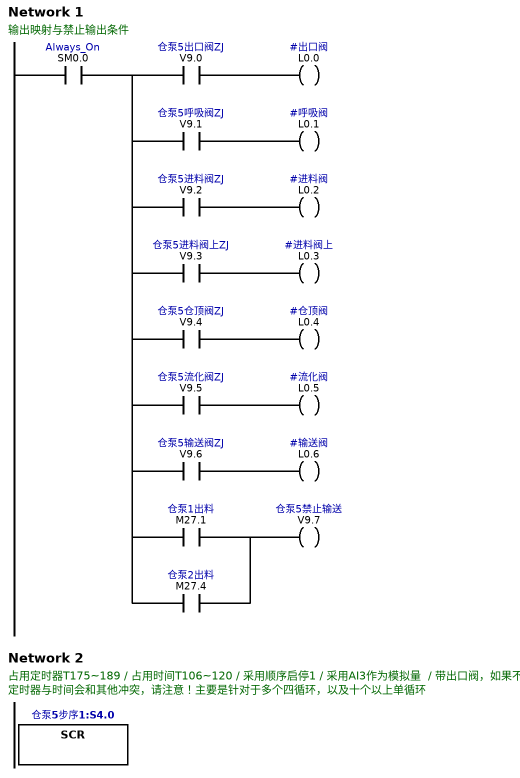
[picture p72: SBR24 networks 1-2]
Network 1
// 输出映射与禁止输出条件
LD     Always_On:SM0.0
LPS
A      仓泵5出口阀ZJ:V9.0
=      #出口阀:L0.0
LRD
A      仓泵5呼吸阀ZJ:V9.1
=      #呼吸阀:L0.1
LRD
A      仓泵5进料阀ZJ:V9.2
=      #进料阀:L0.2
LRD
A      仓泵5进料阀上ZJ:V9.3
=      #进料阀上:L0.3
LRD
A      仓泵5仓顶阀ZJ:V9.4
=      #仓顶阀:L0.4
LRD
A      仓泵5流化阀ZJ:V9.5
=      #流化阀:L0.5
LRD
A      仓泵5输送阀ZJ:V9.6
=      #输送阀:L0.6
LPP
LD     仓泵1出料:M27.1
O      仓泵2出料:M27.4
ALD
=      仓泵5禁止输送:V9.7
Network 2
// 占用定时器T175~189
// 占用时间T106~120
// 采用顺序启停1
// 采用AI3作为模拟量 
// 带出口阀，如果不需要可删除
// 同时仅一个仓泵出料，多需求请改网络5
// 定时器与时间会和其他冲突，请注意！主要是针对于多个四循环，以及十个以上单循环
LSCR   仓泵5步序1:S4.0
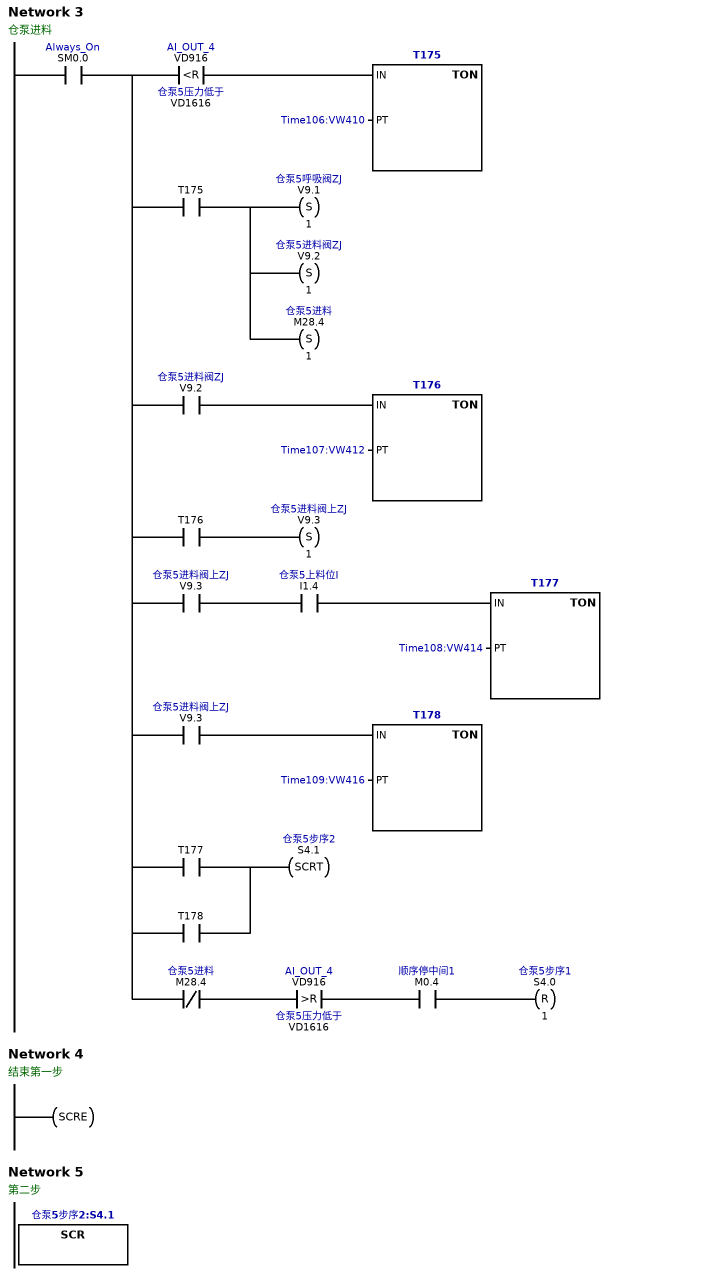
Network 3
// 仓泵进料
LD     Always_On:SM0.0
LPS
AR<    AI_OUT_4:VD916, 仓泵5压力低于:VD1616
TON    T175, Time106:VW410
LRD
A      T175
S      仓泵5呼吸阀ZJ:V9.1, 1
S      仓泵5进料阀ZJ:V9.2, 1
S      仓泵5进料:M28.4, 1
LRD
LPS
A      仓泵5进料阀ZJ:V9.2
TON    T176, Time107:VW412
LRD
A      T176
S      仓泵5进料阀上ZJ:V9.3, 1
LRD
A      仓泵5进料阀上ZJ:V9.3
A      仓泵5上料位I:I1.4
TON    T177, Time108:VW414
LPP
A      仓泵5进料阀上ZJ:V9.3
TON    T178, Time109:VW416
LRD
LD     T177
O      T178
ALD
SCRT   仓泵5步序2:S4.1
LPP
AN     仓泵5进料:M28.4
AR>    AI_OUT_4:VD916, 仓泵5压力低于:VD1616
A      顺序停中间1:M0.4
R      仓泵5步序1:S4.0, 1
Network 4
// 结束第一步
SCRE
Network 5
// 第二步 
LSCR   仓泵5步序2:S4.1
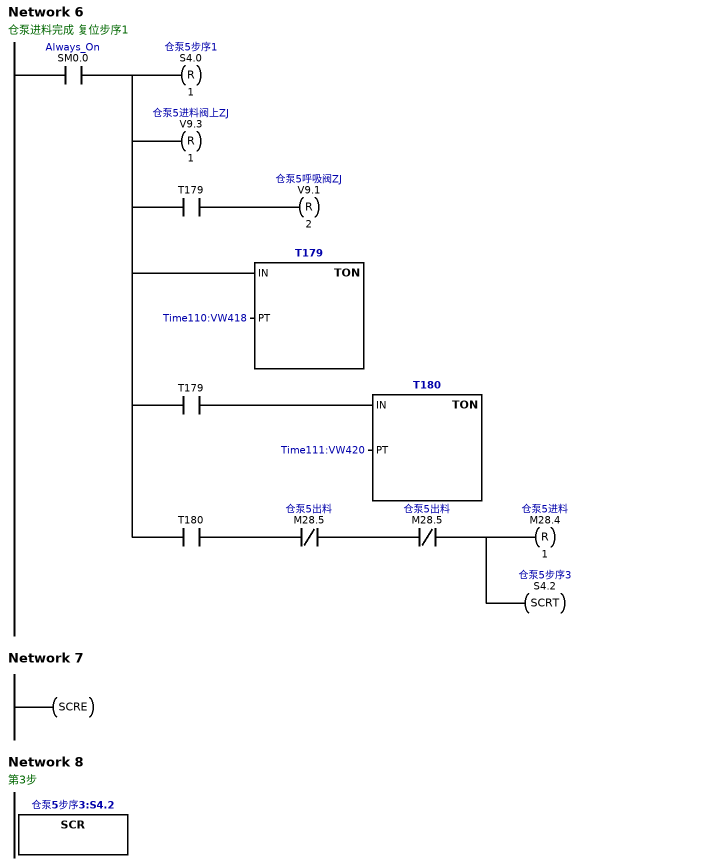
Network 6
// 仓泵进料完成 复位步序1
LD     Always_On:SM0.0
LPS
R      仓泵5步序1:S4.0, 1
R      仓泵5进料阀上ZJ:V9.3, 1
A      T179
R      仓泵5呼吸阀ZJ:V9.1, 2
LRD
TON    T179, Time110:VW418
LRD
A      T179
TON    T180, Time111:VW420
LPP
A      T180
AN     仓泵5出料:M28.5
AN     仓泵5出料:M28.5
R      仓泵5进料:M28.4, 1
SCRT   仓泵5步序3:S4.2
Network 7
SCRE
Network 8
// 第3步 
LSCR   仓泵5步序3:S4.2
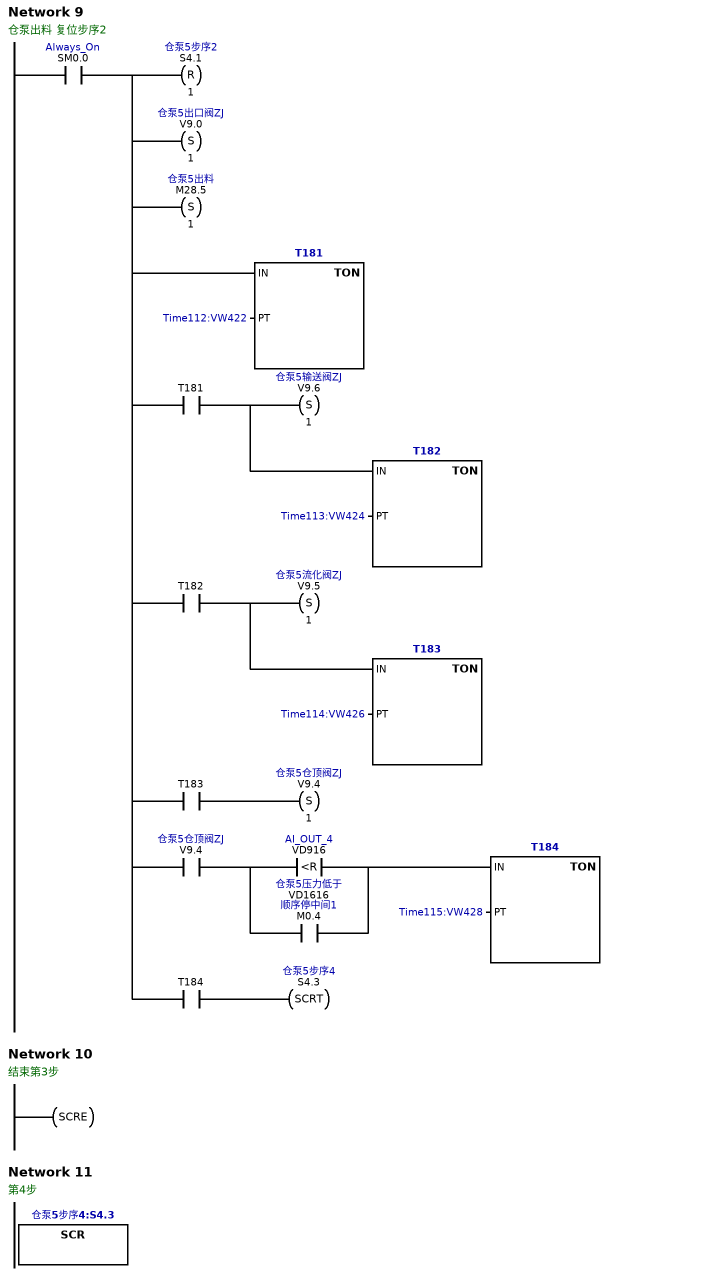
Network 9
// 仓泵出料 复位步序2
LD     Always_On:SM0.0
LPS
R      仓泵5步序2:S4.1, 1
S      仓泵5出口阀ZJ:V9.0, 1
S      仓泵5出料:M28.5, 1
TON    T181, Time112:VW422
A      T181
S      仓泵5输送阀ZJ:V9.6, 1
TON    T182, Time113:VW424
LRD
A      T182
S      仓泵5流化阀ZJ:V9.5, 1
TON    T183, Time114:VW426
LRD
A      T183
S      仓泵5仓顶阀ZJ:V9.4, 1
LRD
A      仓泵5仓顶阀ZJ:V9.4
LDR<   AI_OUT_4:VD916, 仓泵5压力低于:VD1616
O      顺序停中间1:M0.4
ALD
TON    T184, Time115:VW428
LPP
A      T184
SCRT   仓泵5步序4:S4.3
Network 10
// 结束第3步
SCRE
Network 11
// 第4步 
LSCR   仓泵5步序4:S4.3
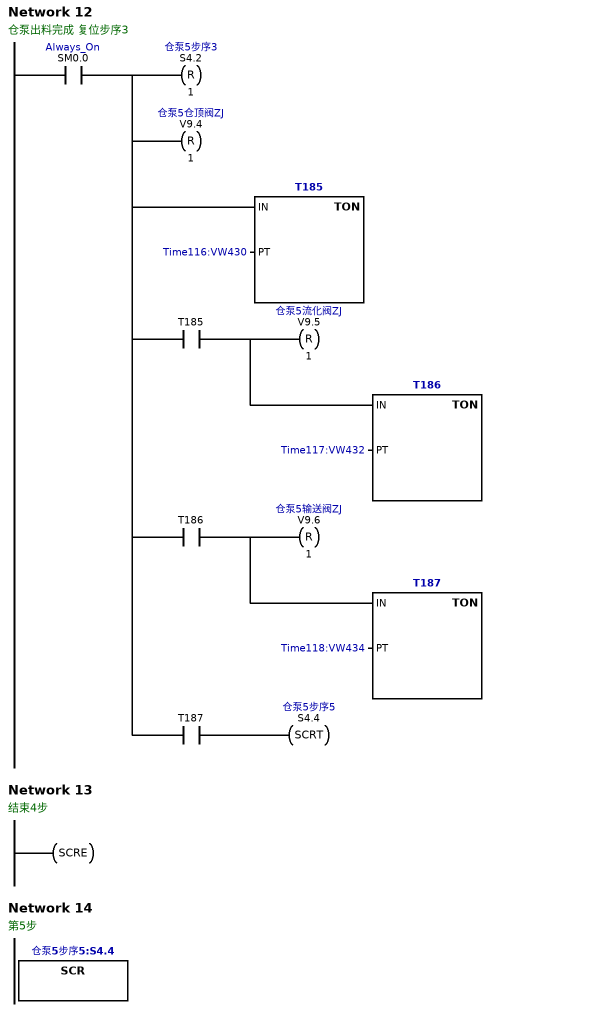
Network 12
// 仓泵出料完成 复位步序3
LD     Always_On:SM0.0
LPS
R      仓泵5步序3:S4.2, 1
R      仓泵5仓顶阀ZJ:V9.4, 1
TON    T185, Time116:VW430
A      T185
R      仓泵5流化阀ZJ:V9.5, 1
TON    T186, Time117:VW432
LRD
A      T186
R      仓泵5输送阀ZJ:V9.6, 1
TON    T187, Time118:VW434
LPP
A      T187
SCRT   仓泵5步序5:S4.4
Network 13
// 结束4步
SCRE
Network 14
// 第5步 
LSCR   仓泵5步序5:S4.4
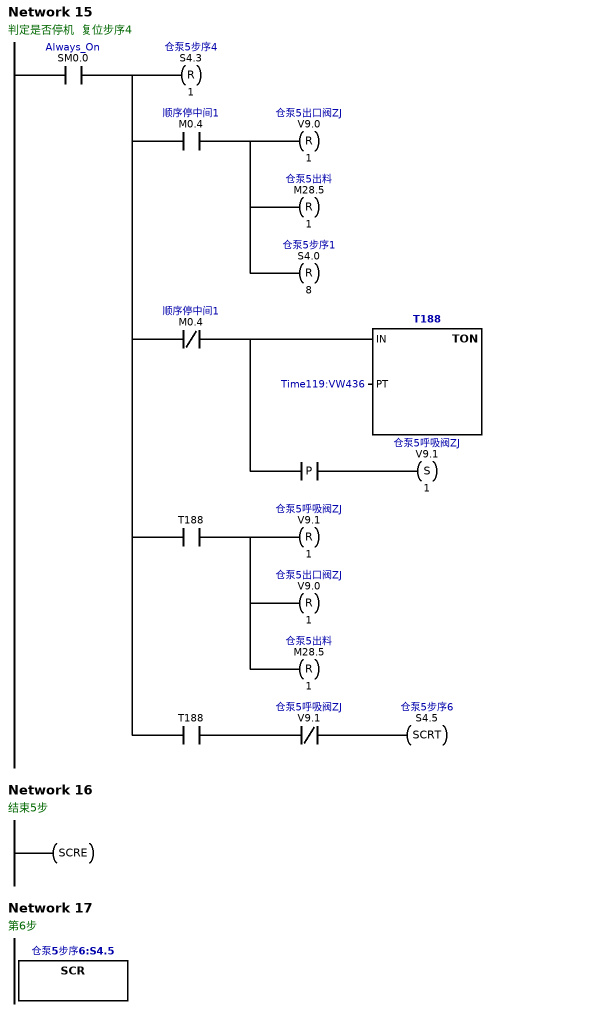
Network 15
// 判定是否停机  复位步序4 
LD     Always_On:SM0.0
LPS
R      仓泵5步序4:S4.3, 1
A      顺序停中间1:M0.4
R      仓泵5出口阀ZJ:V9.0, 1
R      仓泵5出料:M28.5, 1
R      仓泵5步序1:S4.0, 8
LRD
AN     顺序停中间1:M0.4
TON    T188, Time119:VW436
EU
S      仓泵5呼吸阀ZJ:V9.1, 1
LRD
A      T188
R      仓泵5呼吸阀ZJ:V9.1, 1
R      仓泵5出口阀ZJ:V9.0, 1
R      仓泵5出料:M28.5, 1
LPP
A      T188
AN     仓泵5呼吸阀ZJ:V9.1
SCRT   仓泵5步序6:S4.5
Network 16
// 结束5步
SCRE
Network 17
// 第6步 
LSCR   仓泵5步序6:S4.5
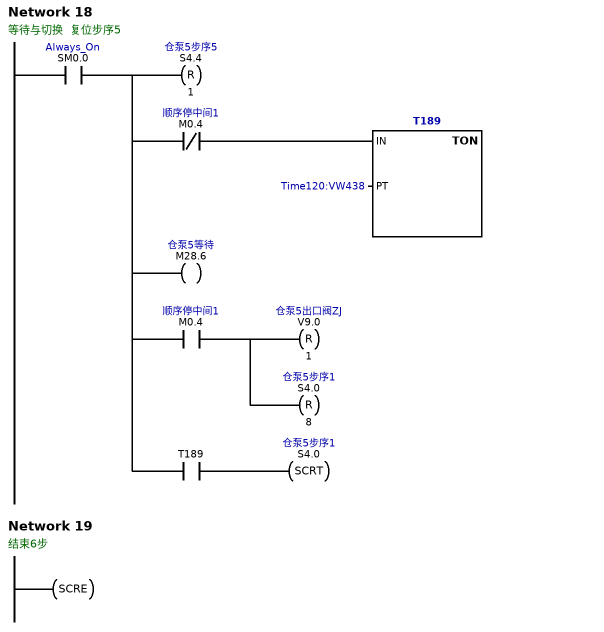
Network 18
// 等待与切换  复位步序5
LD     Always_On:SM0.0
LPS
R      仓泵5步序5:S4.4, 1
AN     顺序停中间1:M0.4
TON    T189, Time120:VW438
LRD
=      仓泵5等待:M28.6
LRD
A      顺序停中间1:M0.4
R      仓泵5出口阀ZJ:V9.0, 1
R      仓泵5步序1:S4.0, 8
LPP
A      T189
SCRT   仓泵5步序1:S4.0
Network 19
// 结束6步
SCRE
END_SUBROUTINE_BLOCK

SUBROUTINE_BLOCK 四除尘器切换:SBR28
TITLE=
VAR_INPUT
IN_T1:BOOL;	// L0.0 
IN_T2:BOOL;	// L0.1 
IN_T3:BOOL;	// L0.2 
IN_T4:BOOL;	// L0.3 
END_VAR
BEGIN
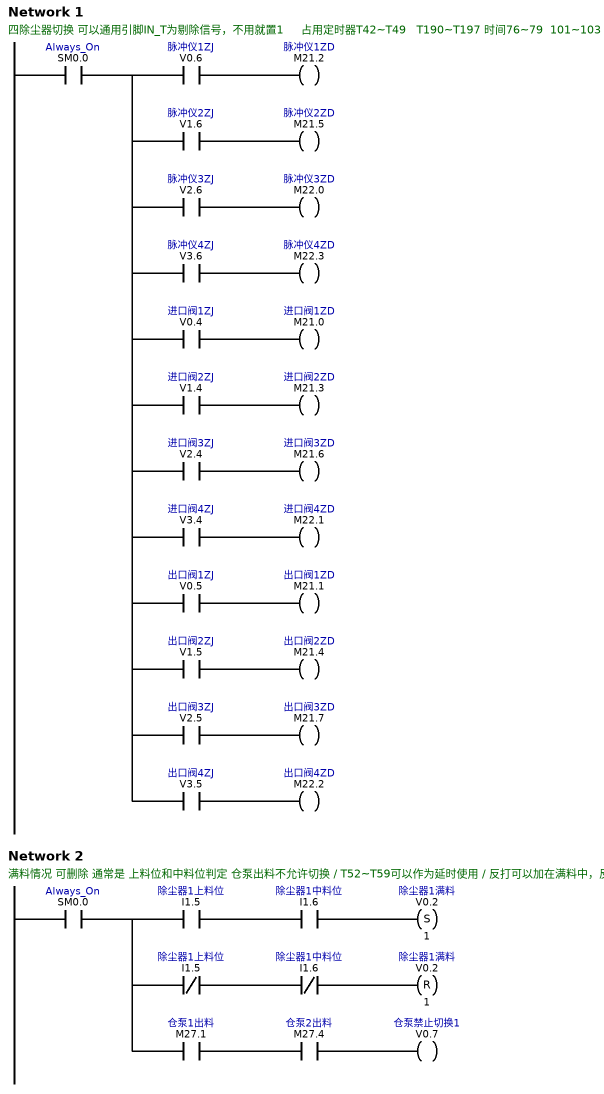
Network 1
// 四除尘器切换 可以通用引脚IN_T为剔除信号，不用就置1     占用定时器T42~T49   T190~T197 时间76~79  101~103 需要对应符号表
// 三除尘器可以沿用此程序，剔除4长通就行 
// 网络1为修改段，主要为输出映射
// 
LD     Always_On:SM0.0
LPS
A      脉冲仪1ZJ:V0.6
=      脉冲仪1ZD:M21.2
LRD
A      脉冲仪2ZJ:V1.6
=      脉冲仪2ZD:M21.5
LRD
A      脉冲仪3ZJ:V2.6
=      脉冲仪3ZD:M22.0
LRD
A      脉冲仪4ZJ:V3.6
=      脉冲仪4ZD:M22.3
LRD
A      进口阀1ZJ:V0.4
=      进口阀1ZD:M21.0
LRD
A      进口阀2ZJ:V1.4
=      进口阀2ZD:M21.3
LRD
A      进口阀3ZJ:V2.4
=      进口阀3ZD:M21.6
LRD
A      进口阀4ZJ:V3.4
=      进口阀4ZD:M22.1
LRD
A      出口阀1ZJ:V0.5
=      出口阀1ZD:M21.1
LRD
A      出口阀2ZJ:V1.5
=      出口阀2ZD:M21.4
LRD
A      出口阀3ZJ:V2.5
=      出口阀3ZD:M21.7
LPP
A      出口阀4ZJ:V3.5
=      出口阀4ZD:M22.2
Network 2
// 满料情况 可删除 通常是 上料位和中料位判定 仓泵出料不允许切换
// T52~T59可以作为延时使用
// 反打可以加在满料中，反打时禁止除尘器进料
LD     Always_On:SM0.0
LPS
A      除尘器1上料位:I1.5
A      除尘器1中料位:I1.6
S      除尘器1满料:V0.2, 1
LRD
AN     除尘器1上料位:I1.5
AN     除尘器1中料位:I1.6
R      除尘器1满料:V0.2, 1
LPP
A      仓泵1出料:M27.1
A      仓泵2出料:M27.4
=      仓泵禁止切换1:V0.7
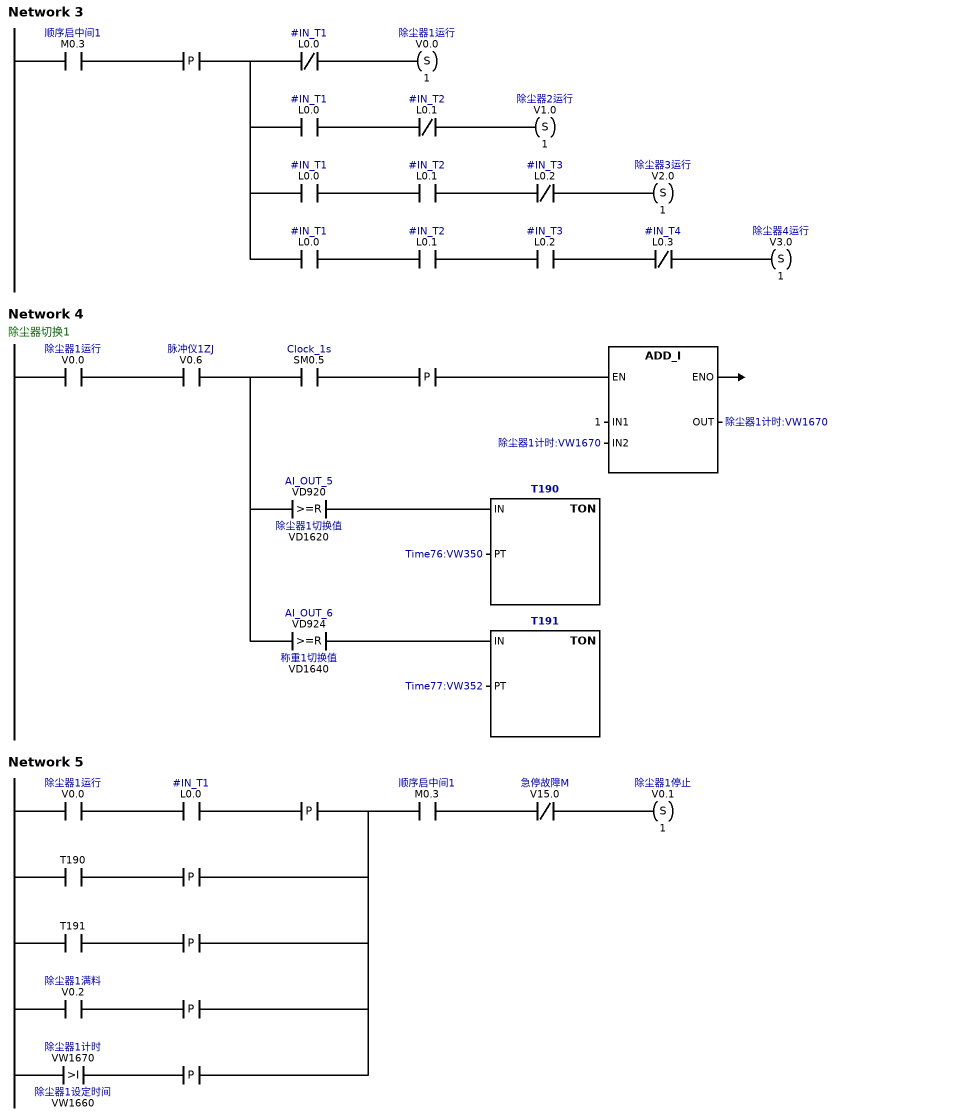
Network 3
//   
// 
LD     顺序启中间1:M0.3
EU
LPS
AN     #IN_T1:L0.0
S      除尘器1运行:V0.0, 1
LRD
A      #IN_T1:L0.0
AN     #IN_T2:L0.1
S      除尘器2运行:V1.0, 1
LRD
A      #IN_T1:L0.0
A      #IN_T2:L0.1
AN     #IN_T3:L0.2
S      除尘器3运行:V2.0, 1
LPP
A      #IN_T1:L0.0
A      #IN_T2:L0.1
A      #IN_T3:L0.2
AN     #IN_T4:L0.3
S      除尘器4运行:V3.0, 1
Network 4
// 除尘器切换1
LD     除尘器1运行:V0.0
A      脉冲仪1ZJ:V0.6
LPS
A      Clock_1s:SM0.5
EU
+I     1, 除尘器1计时:VW1670
LRD
AR>=   AI_OUT_5:VD920, 除尘器1切换值:VD1620
TON    T190, Time76:VW350
LPP
AR>=   AI_OUT_6:VD924, 称重1切换值:VD1640
TON    T191, Time77:VW352
Network 5
LD     除尘器1运行:V0.0
A      #IN_T1:L0.0
EU
LD     T190
EU
OLD
LD     T191
EU
OLD
LD     除尘器1满料:V0.2
EU
OLD
LDW>   除尘器1计时:VW1670, 除尘器1设定时间:VW1660
EU
OLD
A      顺序启中间1:M0.3
AN     急停故障M:V15.0
S      除尘器1停止:V0.1, 1
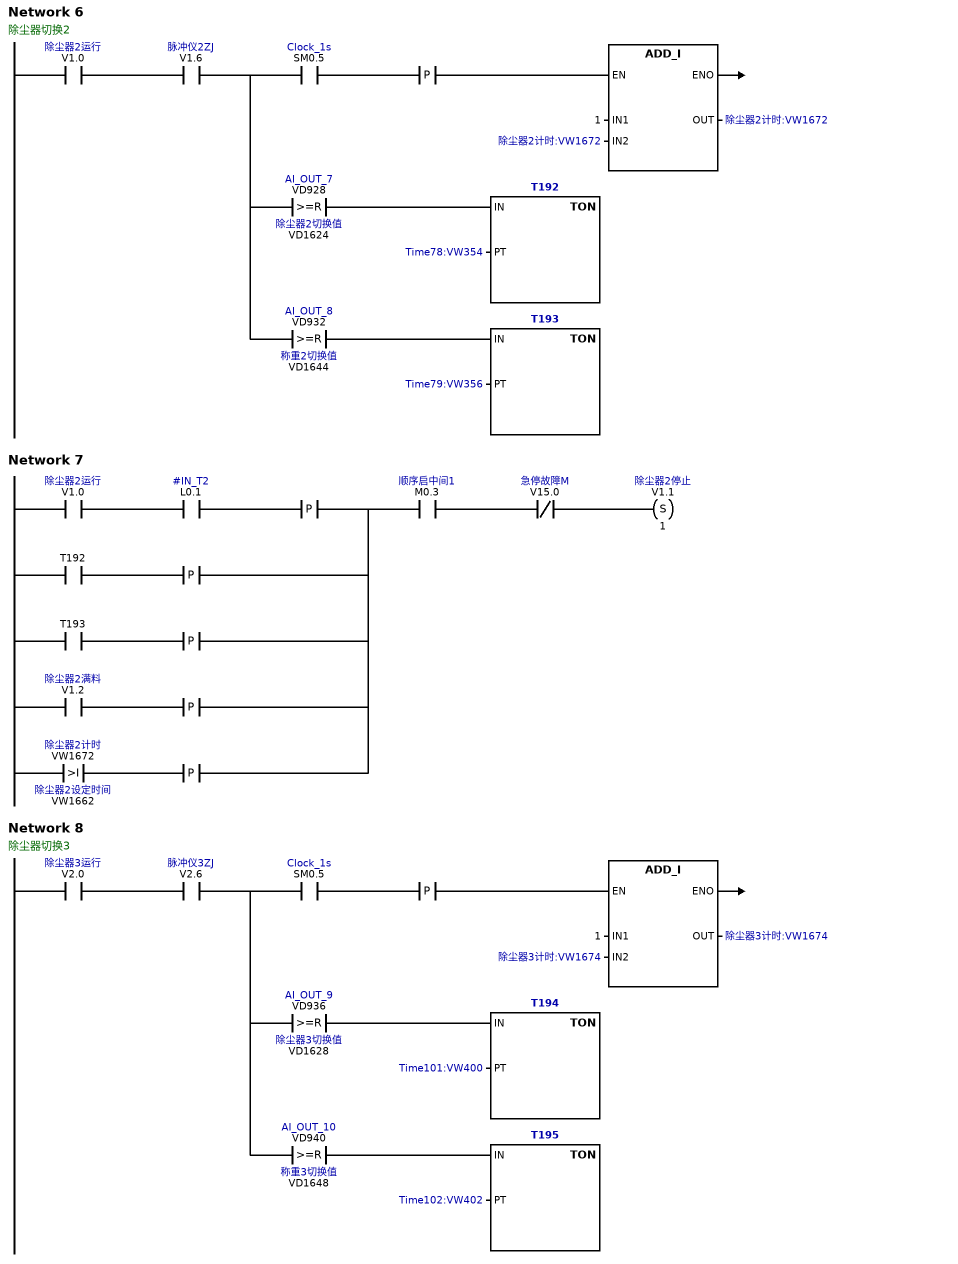
Network 6
// 除尘器切换2
LD     除尘器2运行:V1.0
A      脉冲仪2ZJ:V1.6
LPS
A      Clock_1s:SM0.5
EU
+I     1, 除尘器2计时:VW1672
LRD
AR>=   AI_OUT_7:VD928, 除尘器2切换值:VD1624
TON    T192, Time78:VW354
LPP
AR>=   AI_OUT_8:VD932, 称重2切换值:VD1644
TON    T193, Time79:VW356
Network 7
LD     除尘器2运行:V1.0
A      #IN_T2:L0.1
EU
LD     T192
EU
OLD
LD     T193
EU
OLD
LD     除尘器2满料:V1.2
EU
OLD
LDW>   除尘器2计时:VW1672, 除尘器2设定时间:VW1662
EU
OLD
A      顺序启中间1:M0.3
AN     急停故障M:V15.0
S      除尘器2停止:V1.1, 1
Network 8
// 除尘器切换3
LD     除尘器3运行:V2.0
A      脉冲仪3ZJ:V2.6
LPS
A      Clock_1s:SM0.5
EU
+I     1, 除尘器3计时:VW1674
LRD
AR>=   AI_OUT_9:VD936, 除尘器3切换值:VD1628
TON    T194, Time101:VW400
LPP
AR>=   AI_OUT_10:VD940, 称重3切换值:VD1648
TON    T195, Time102:VW402
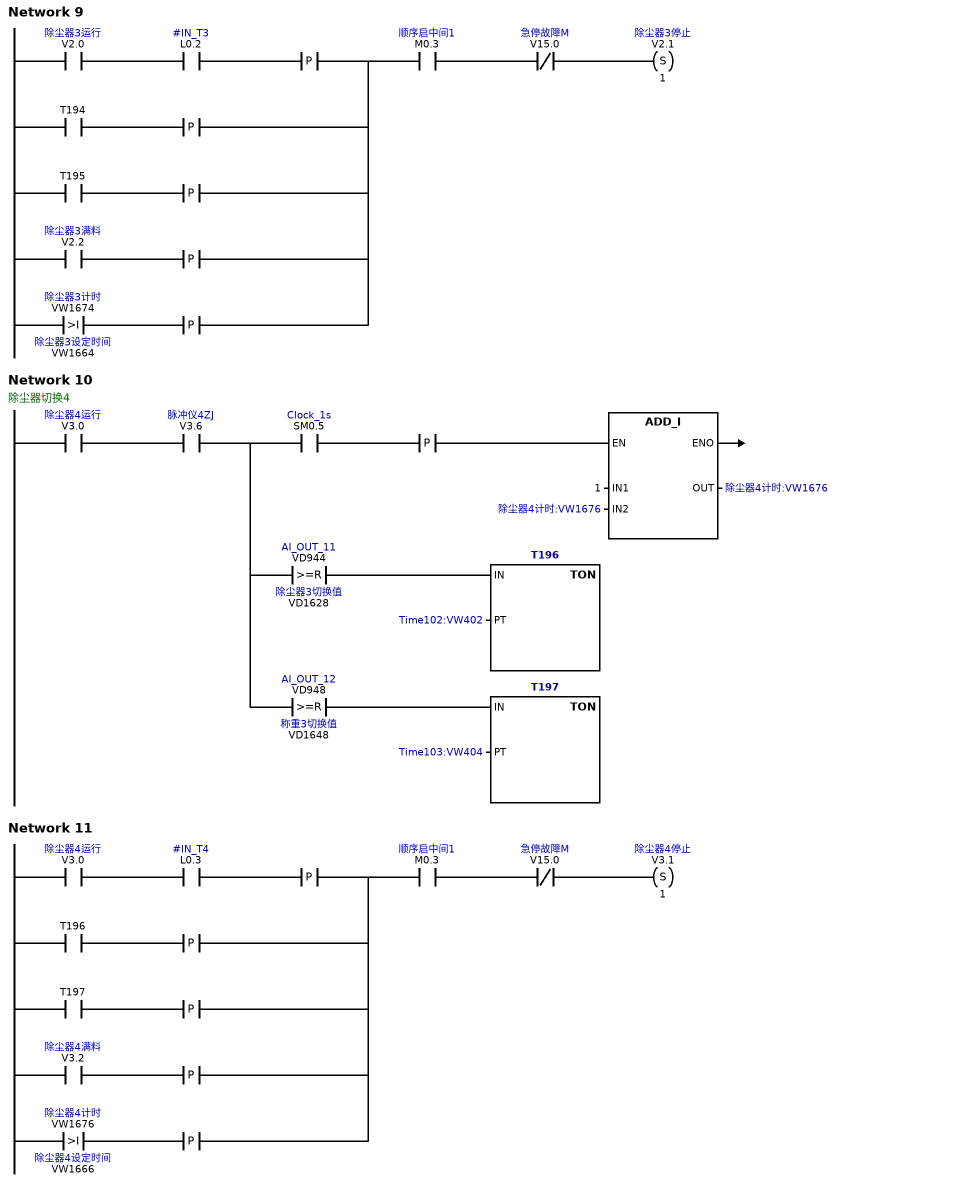
Network 9
LD     除尘器3运行:V2.0
A      #IN_T3:L0.2
EU
LD     T194
EU
OLD
LD     T195
EU
OLD
LD     除尘器3满料:V2.2
EU
OLD
LDW>   除尘器3计时:VW1674, 除尘器3设定时间:VW1664
EU
OLD
A      顺序启中间1:M0.3
AN     急停故障M:V15.0
S      除尘器3停止:V2.1, 1
Network 10
// 除尘器切换4
LD     除尘器4运行:V3.0
A      脉冲仪4ZJ:V3.6
LPS
A      Clock_1s:SM0.5
EU
+I     1, 除尘器4计时:VW1676
LRD
AR>=   AI_OUT_11:VD944, 除尘器3切换值:VD1628
TON    T196, Time102:VW402
LPP
AR>=   AI_OUT_12:VD948, 称重3切换值:VD1648
TON    T197, Time103:VW404
Network 11
LD     除尘器4运行:V3.0
A      #IN_T4:L0.3
EU
LD     T196
EU
OLD
LD     T197
EU
OLD
LD     除尘器4满料:V3.2
EU
OLD
LDW>   除尘器4计时:VW1676, 除尘器4设定时间:VW1666
EU
OLD
A      顺序启中间1:M0.3
AN     急停故障M:V15.0
S      除尘器4停止:V3.1, 1
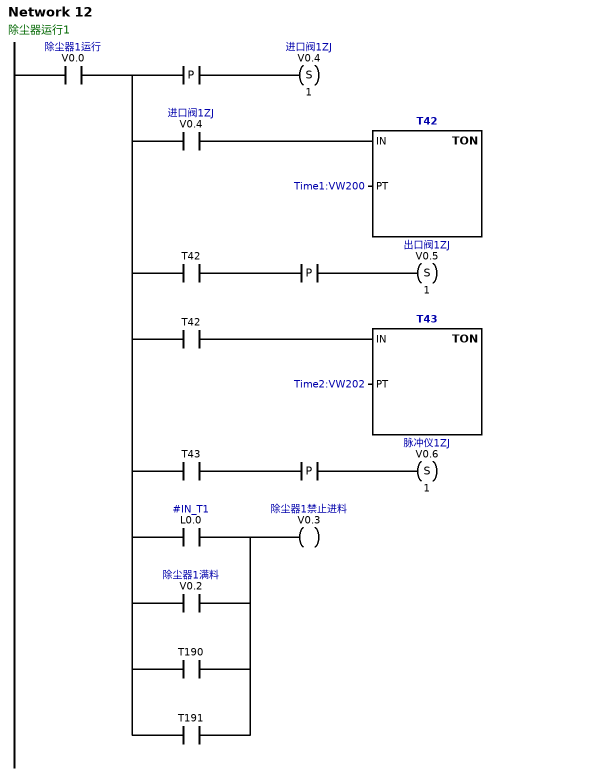
Network 12
// 除尘器运行1
LD     除尘器1运行:V0.0
LPS
EU
S      进口阀1ZJ:V0.4, 1
LRD
A      进口阀1ZJ:V0.4
TON    T42, Time1:VW200
LRD
A      T42
EU
S      出口阀1ZJ:V0.5, 1
LRD
A      T42
TON    T43, Time2:VW202
LRD
A      T43
EU
S      脉冲仪1ZJ:V0.6, 1
LPP
LD     #IN_T1:L0.0
O      除尘器1满料:V0.2
O      T190
O      T191
ALD
=      除尘器1禁止进料:V0.3
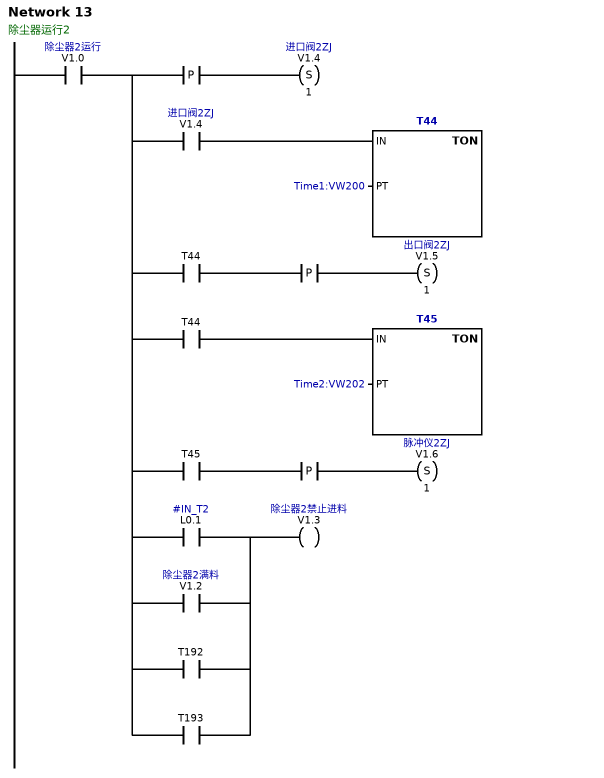
Network 13
// 除尘器运行2
LD     除尘器2运行:V1.0
LPS
EU
S      进口阀2ZJ:V1.4, 1
LRD
A      进口阀2ZJ:V1.4
TON    T44, Time1:VW200
LRD
A      T44
EU
S      出口阀2ZJ:V1.5, 1
LRD
A      T44
TON    T45, Time2:VW202
LRD
A      T45
EU
S      脉冲仪2ZJ:V1.6, 1
LPP
LD     #IN_T2:L0.1
O      除尘器2满料:V1.2
O      T192
O      T193
ALD
=      除尘器2禁止进料:V1.3
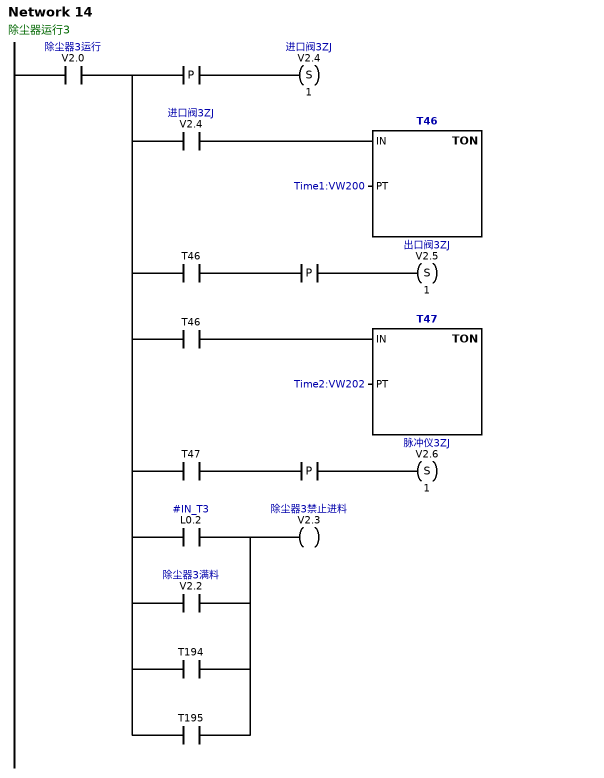
Network 14
// 除尘器运行3
LD     除尘器3运行:V2.0
LPS
EU
S      进口阀3ZJ:V2.4, 1
LRD
A      进口阀3ZJ:V2.4
TON    T46, Time1:VW200
LRD
A      T46
EU
S      出口阀3ZJ:V2.5, 1
LRD
A      T46
TON    T47, Time2:VW202
LRD
A      T47
EU
S      脉冲仪3ZJ:V2.6, 1
LPP
LD     #IN_T3:L0.2
O      除尘器3满料:V2.2
O      T194
O      T195
ALD
=      除尘器3禁止进料:V2.3
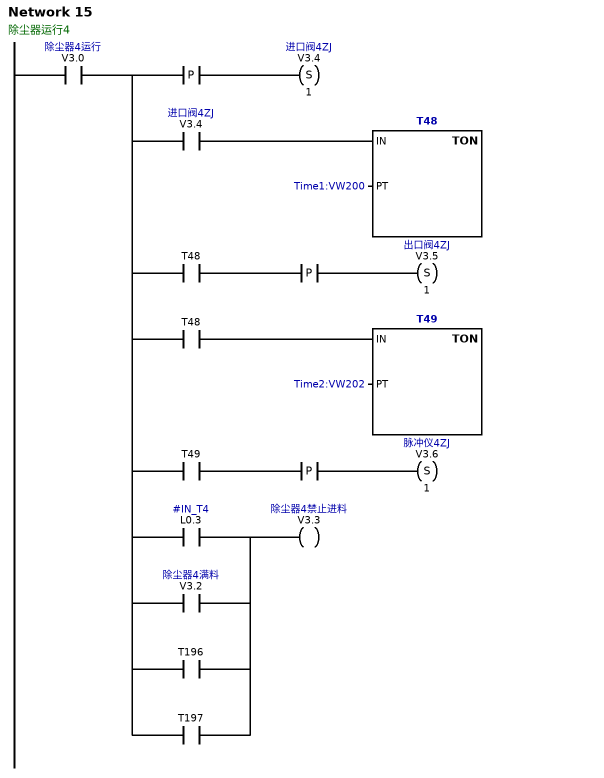
Network 15
// 除尘器运行4
LD     除尘器4运行:V3.0
LPS
EU
S      进口阀4ZJ:V3.4, 1
LRD
A      进口阀4ZJ:V3.4
TON    T48, Time1:VW200
LRD
A      T48
EU
S      出口阀4ZJ:V3.5, 1
LRD
A      T48
TON    T49, Time2:VW202
LRD
A      T49
EU
S      脉冲仪4ZJ:V3.6, 1
LPP
LD     #IN_T4:L0.3
O      除尘器4满料:V3.2
O      T196
O      T197
ALD
=      除尘器4禁止进料:V3.3
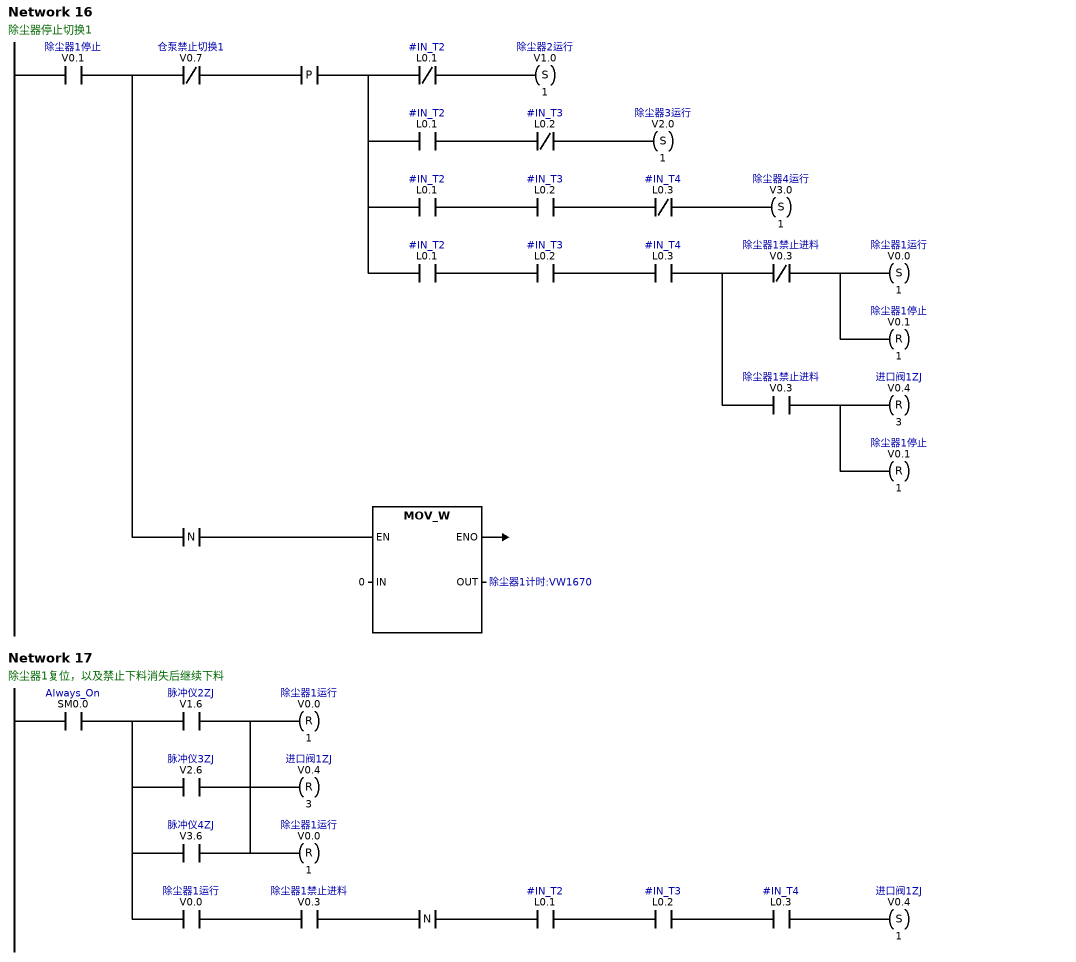
Network 16
// 除尘器停止切换1
LD     除尘器1停止:V0.1
LPS
AN     仓泵禁止切换1:V0.7
EU
LPS
AN     #IN_T2:L0.1
S      除尘器2运行:V1.0, 1
LRD
A      #IN_T2:L0.1
AN     #IN_T3:L0.2
S      除尘器3运行:V2.0, 1
LRD
A      #IN_T2:L0.1
A      #IN_T3:L0.2
AN     #IN_T4:L0.3
S      除尘器4运行:V3.0, 1
LPP
A      #IN_T2:L0.1
A      #IN_T3:L0.2
A      #IN_T4:L0.3
LPS
AN     除尘器1禁止进料:V0.3
S      除尘器1运行:V0.0, 1
R      除尘器1停止:V0.1, 1
LPP
A      除尘器1禁止进料:V0.3
R      进口阀1ZJ:V0.4, 3
R      除尘器1停止:V0.1, 1
LPP
ED
MOVW   0, 除尘器1计时:VW1670
Network 17
// 除尘器1复位，以及禁止下料消失后继续下料
LD     Always_On:SM0.0
LPS
LD     脉冲仪2ZJ:V1.6
O      脉冲仪3ZJ:V2.6
O      脉冲仪4ZJ:V3.6
ALD
R      除尘器1运行:V0.0, 1
R      进口阀1ZJ:V0.4, 3
R      除尘器1运行:V0.0, 1
LPP
A      除尘器1运行:V0.0
A      除尘器1禁止进料:V0.3
ED
A      #IN_T2:L0.1
A      #IN_T3:L0.2
A      #IN_T4:L0.3
S      进口阀1ZJ:V0.4, 1
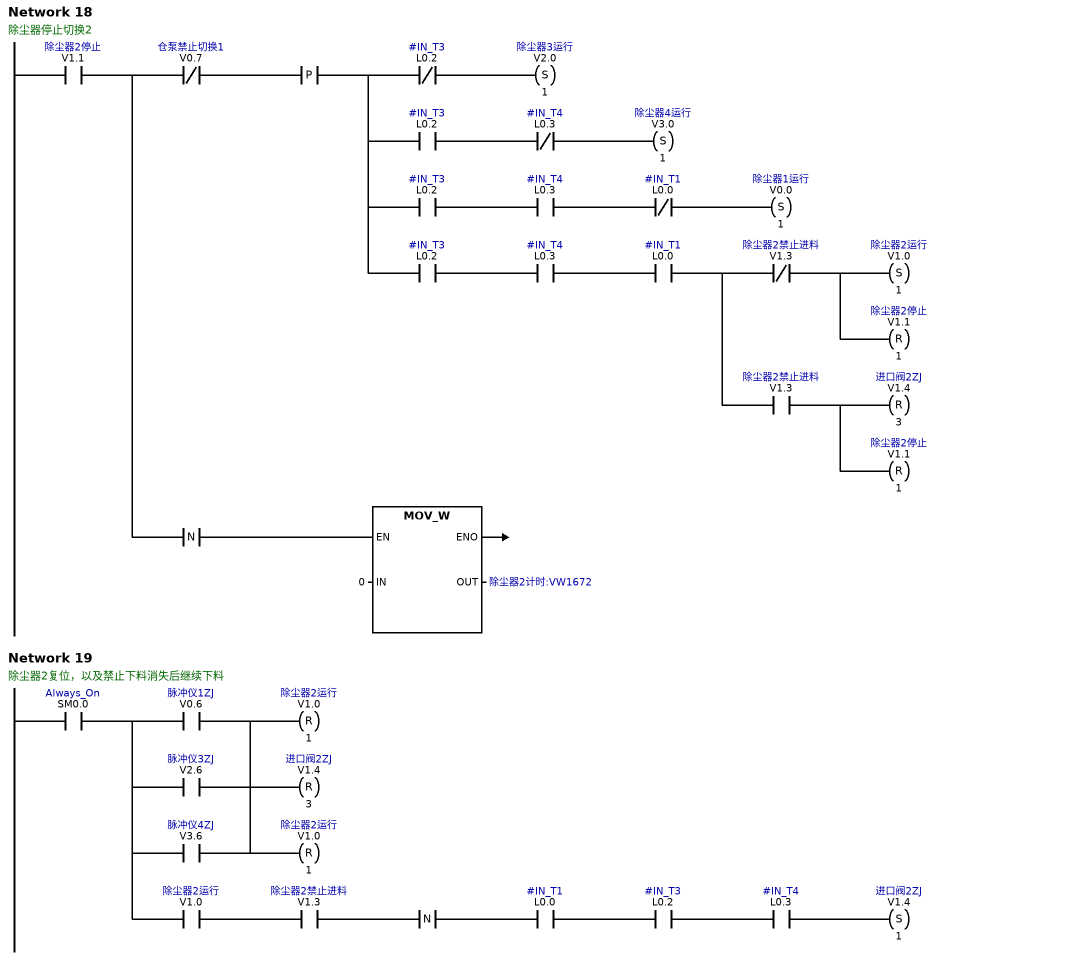
Network 18
// 除尘器停止切换2
LD     除尘器2停止:V1.1
LPS
AN     仓泵禁止切换1:V0.7
EU
LPS
AN     #IN_T3:L0.2
S      除尘器3运行:V2.0, 1
LRD
A      #IN_T3:L0.2
AN     #IN_T4:L0.3
S      除尘器4运行:V3.0, 1
LRD
A      #IN_T3:L0.2
A      #IN_T4:L0.3
AN     #IN_T1:L0.0
S      除尘器1运行:V0.0, 1
LPP
A      #IN_T3:L0.2
A      #IN_T4:L0.3
A      #IN_T1:L0.0
LPS
AN     除尘器2禁止进料:V1.3
S      除尘器2运行:V1.0, 1
R      除尘器2停止:V1.1, 1
LPP
A      除尘器2禁止进料:V1.3
R      进口阀2ZJ:V1.4, 3
R      除尘器2停止:V1.1, 1
LPP
ED
MOVW   0, 除尘器2计时:VW1672
Network 19
// 除尘器2复位，以及禁止下料消失后继续下料
LD     Always_On:SM0.0
LPS
LD     脉冲仪1ZJ:V0.6
O      脉冲仪3ZJ:V2.6
O      脉冲仪4ZJ:V3.6
ALD
R      除尘器2运行:V1.0, 1
R      进口阀2ZJ:V1.4, 3
R      除尘器2运行:V1.0, 1
LPP
A      除尘器2运行:V1.0
A      除尘器2禁止进料:V1.3
ED
A      #IN_T1:L0.0
A      #IN_T3:L0.2
A      #IN_T4:L0.3
S      进口阀2ZJ:V1.4, 1
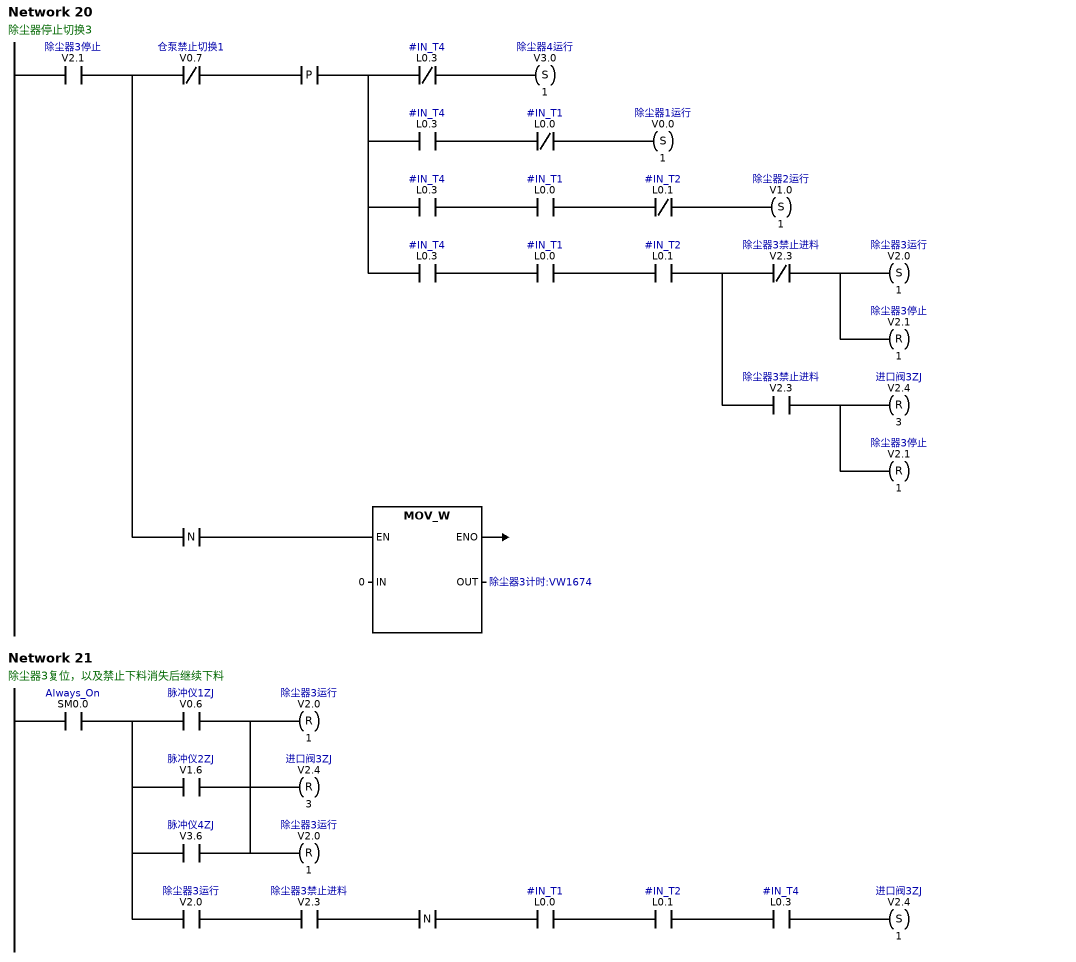
Network 20
// 除尘器停止切换3
LD     除尘器3停止:V2.1
LPS
AN     仓泵禁止切换1:V0.7
EU
LPS
AN     #IN_T4:L0.3
S      除尘器4运行:V3.0, 1
LRD
A      #IN_T4:L0.3
AN     #IN_T1:L0.0
S      除尘器1运行:V0.0, 1
LRD
A      #IN_T4:L0.3
A      #IN_T1:L0.0
AN     #IN_T2:L0.1
S      除尘器2运行:V1.0, 1
LPP
A      #IN_T4:L0.3
A      #IN_T1:L0.0
A      #IN_T2:L0.1
LPS
AN     除尘器3禁止进料:V2.3
S      除尘器3运行:V2.0, 1
R      除尘器3停止:V2.1, 1
LPP
A      除尘器3禁止进料:V2.3
R      进口阀3ZJ:V2.4, 3
R      除尘器3停止:V2.1, 1
LPP
ED
MOVW   0, 除尘器3计时:VW1674
Network 21
// 除尘器3复位，以及禁止下料消失后继续下料
LD     Always_On:SM0.0
LPS
LD     脉冲仪1ZJ:V0.6
O      脉冲仪2ZJ:V1.6
O      脉冲仪4ZJ:V3.6
ALD
R      除尘器3运行:V2.0, 1
R      进口阀3ZJ:V2.4, 3
R      除尘器3运行:V2.0, 1
LPP
A      除尘器3运行:V2.0
A      除尘器3禁止进料:V2.3
ED
A      #IN_T1:L0.0
A      #IN_T2:L0.1
A      #IN_T4:L0.3
S      进口阀3ZJ:V2.4, 1
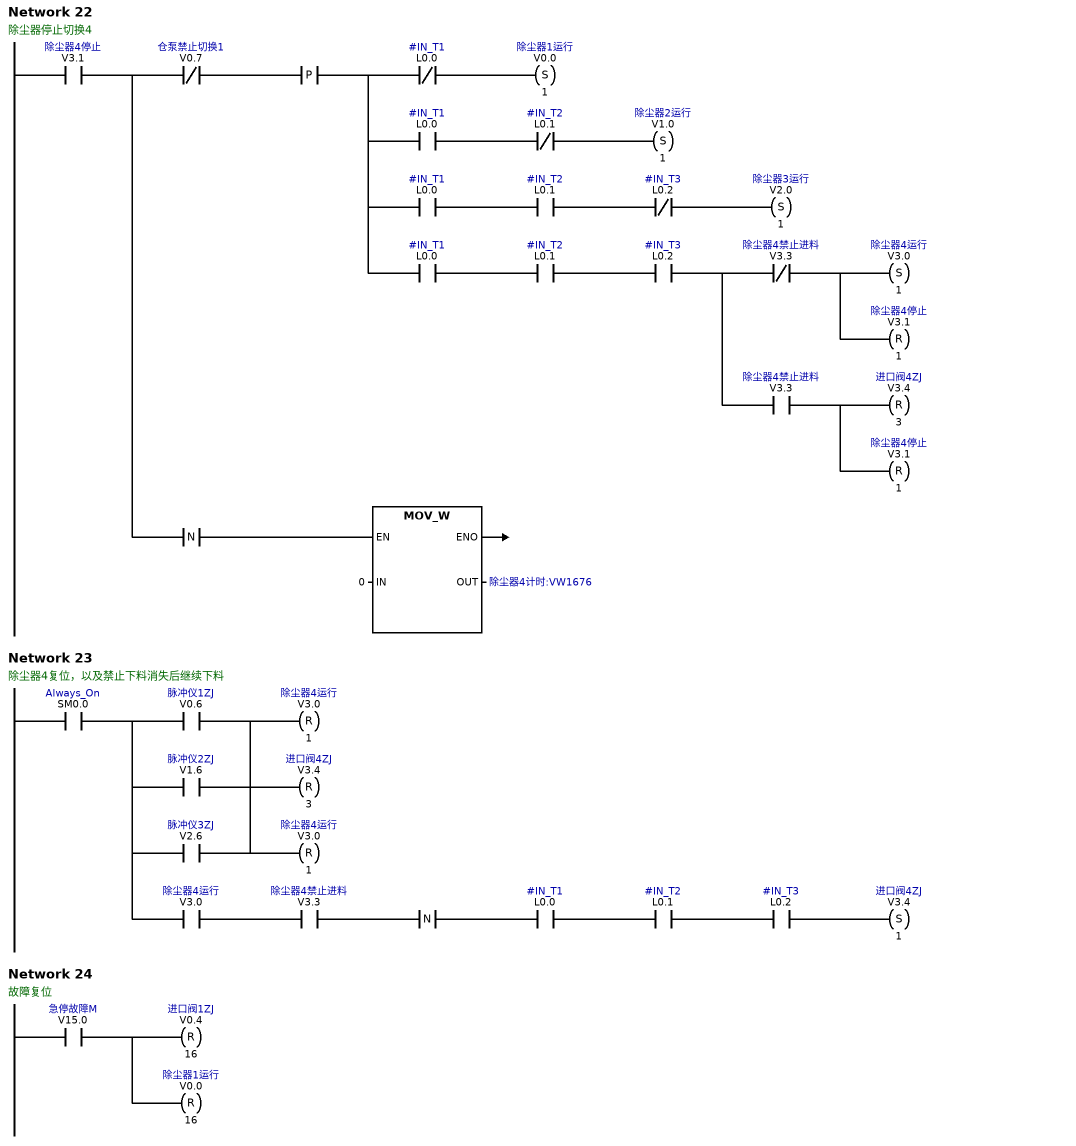
Network 22
// 除尘器停止切换4
LD     除尘器4停止:V3.1
LPS
AN     仓泵禁止切换1:V0.7
EU
LPS
AN     #IN_T1:L0.0
S      除尘器1运行:V0.0, 1
LRD
A      #IN_T1:L0.0
AN     #IN_T2:L0.1
S      除尘器2运行:V1.0, 1
LRD
A      #IN_T1:L0.0
A      #IN_T2:L0.1
AN     #IN_T3:L0.2
S      除尘器3运行:V2.0, 1
LPP
A      #IN_T1:L0.0
A      #IN_T2:L0.1
A      #IN_T3:L0.2
LPS
AN     除尘器4禁止进料:V3.3
S      除尘器4运行:V3.0, 1
R      除尘器4停止:V3.1, 1
LPP
A      除尘器4禁止进料:V3.3
R      进口阀4ZJ:V3.4, 3
R      除尘器4停止:V3.1, 1
LPP
ED
MOVW   0, 除尘器4计时:VW1676
Network 23
// 除尘器4复位，以及禁止下料消失后继续下料
LD     Always_On:SM0.0
LPS
LD     脉冲仪1ZJ:V0.6
O      脉冲仪2ZJ:V1.6
O      脉冲仪3ZJ:V2.6
ALD
R      除尘器4运行:V3.0, 1
R      进口阀4ZJ:V3.4, 3
R      除尘器4运行:V3.0, 1
LPP
A      除尘器4运行:V3.0
A      除尘器4禁止进料:V3.3
ED
A      #IN_T1:L0.0
A      #IN_T2:L0.1
A      #IN_T3:L0.2
S      进口阀4ZJ:V3.4, 1
Network 24
// 故障复位
LD     急停故障M:V15.0
R      进口阀1ZJ:V0.4, 16
R      除尘器1运行:V0.0, 16
END_SUBROUTINE_BLOCK

SUBROUTINE_BLOCK 三除尘器双系统:SBR29
TITLE=
VAR_INPUT
IN_T1:BOOL;	// L0.0 
IN_T2:BOOL;	// L0.1 
IN_T3:BOOL;	// L0.2 
IN_T4:BOOL;	// L0.3 
END_VAR
VAR_OUTPUT
OUT_MC1:BOOL;	// L0.4 
OUT_MC2:BOOL;	// L0.5 
OUT_MC3:BOOL;	// L0.6 
OUT_MC4:BOOL;	// L0.7 
END_VAR
BEGIN
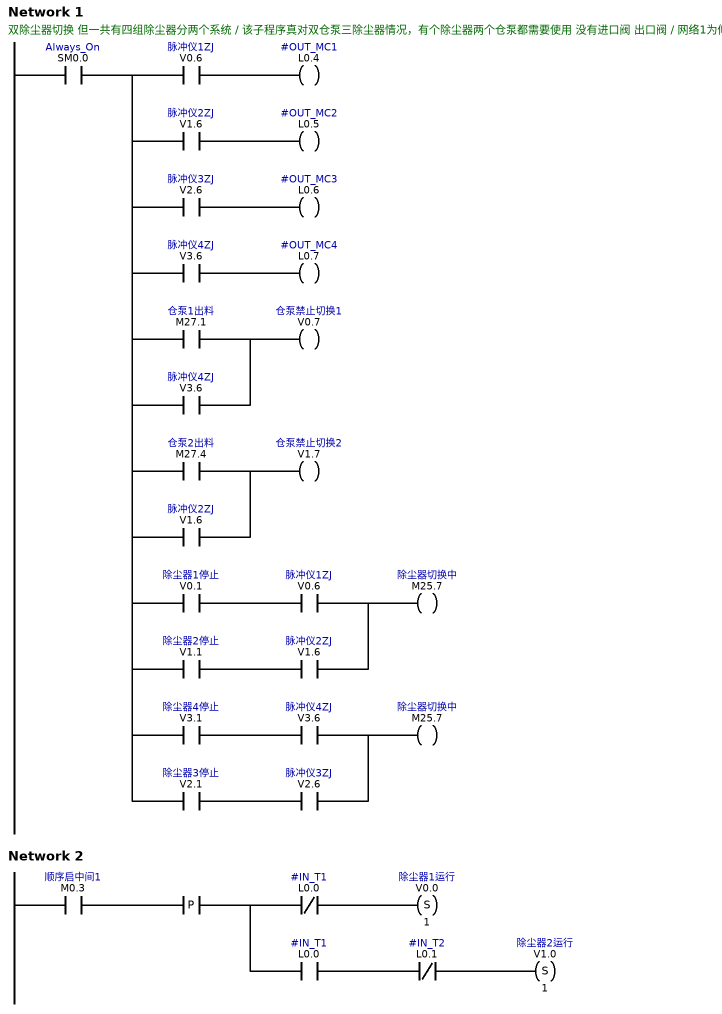
Network 1
// 双除尘器切换 但一共有四组除尘器分两个系统
// 该子程序真对双仓泵三除尘器情况，有个除尘器两个仓泵都需要使用 没有进口阀 出口阀
// 网络1为修改段，主要为输出映射
// 
LD     Always_On:SM0.0
LPS
A      脉冲仪1ZJ:V0.6
=      #OUT_MC1:L0.4
LRD
A      脉冲仪2ZJ:V1.6
=      #OUT_MC2:L0.5
LRD
A      脉冲仪3ZJ:V2.6
=      #OUT_MC3:L0.6
LRD
A      脉冲仪4ZJ:V3.6
=      #OUT_MC4:L0.7
LRD
LD     仓泵1出料:M27.1
O      脉冲仪4ZJ:V3.6
ALD
=      仓泵禁止切换1:V0.7
LRD
LD     仓泵2出料:M27.4
O      脉冲仪2ZJ:V1.6
ALD
=      仓泵禁止切换2:V1.7
LRD
LD     除尘器1停止:V0.1
A      脉冲仪1ZJ:V0.6
LD     除尘器2停止:V1.1
A      脉冲仪2ZJ:V1.6
OLD
ALD
=      除尘器切换中:M25.7
LPP
LD     除尘器4停止:V3.1
A      脉冲仪4ZJ:V3.6
LD     除尘器3停止:V2.1
A      脉冲仪3ZJ:V2.6
OLD
ALD
=      除尘器切换中:M25.7
Network 2
//   
// 
LD     顺序启中间1:M0.3
EU
LPS
AN     #IN_T1:L0.0
S      除尘器1运行:V0.0, 1
LPP
A      #IN_T1:L0.0
AN     #IN_T2:L0.1
S      除尘器2运行:V1.0, 1
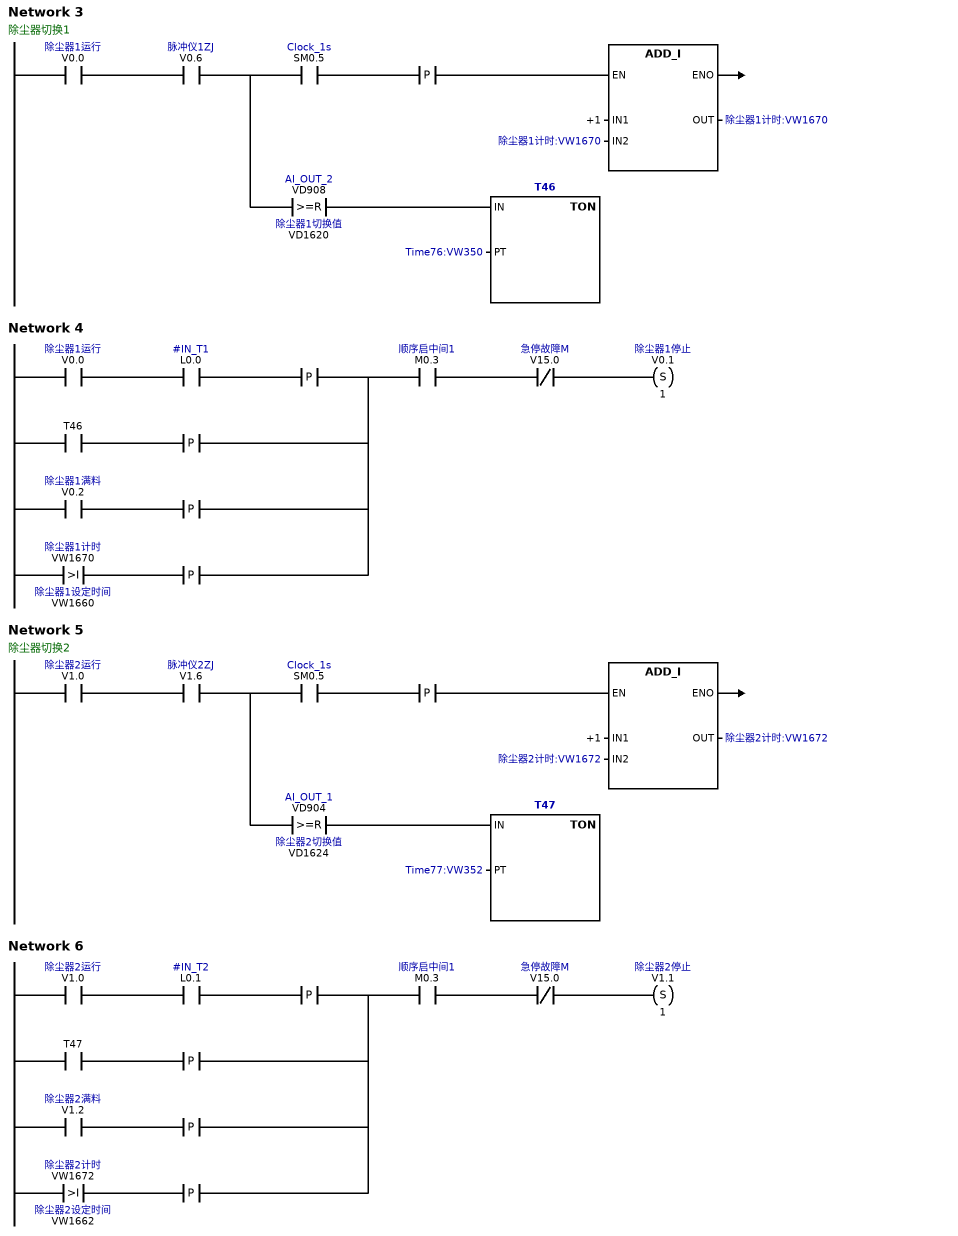
Network 3
// 除尘器切换1
LD     除尘器1运行:V0.0
A      脉冲仪1ZJ:V0.6
LPS
A      Clock_1s:SM0.5
EU
+I     +1, 除尘器1计时:VW1670
LPP
AR>=   AI_OUT_2:VD908, 除尘器1切换值:VD1620
TON    T46, Time76:VW350
Network 4
LD     除尘器1运行:V0.0
A      #IN_T1:L0.0
EU
LD     T46
EU
OLD
LD     除尘器1满料:V0.2
EU
OLD
LDW>   除尘器1计时:VW1670, 除尘器1设定时间:VW1660
EU
OLD
A      顺序启中间1:M0.3
AN     急停故障M:V15.0
S      除尘器1停止:V0.1, 1
Network 5
// 除尘器切换2
LD     除尘器2运行:V1.0
A      脉冲仪2ZJ:V1.6
LPS
A      Clock_1s:SM0.5
EU
+I     +1, 除尘器2计时:VW1672
LPP
AR>=   AI_OUT_1:VD904, 除尘器2切换值:VD1624
TON    T47, Time77:VW352
Network 6
LD     除尘器2运行:V1.0
A      #IN_T2:L0.1
EU
LD     T47
EU
OLD
LD     除尘器2满料:V1.2
EU
OLD
LDW>   除尘器2计时:VW1672, 除尘器2设定时间:VW1662
EU
OLD
A      顺序启中间1:M0.3
AN     急停故障M:V15.0
S      除尘器2停止:V1.1, 1
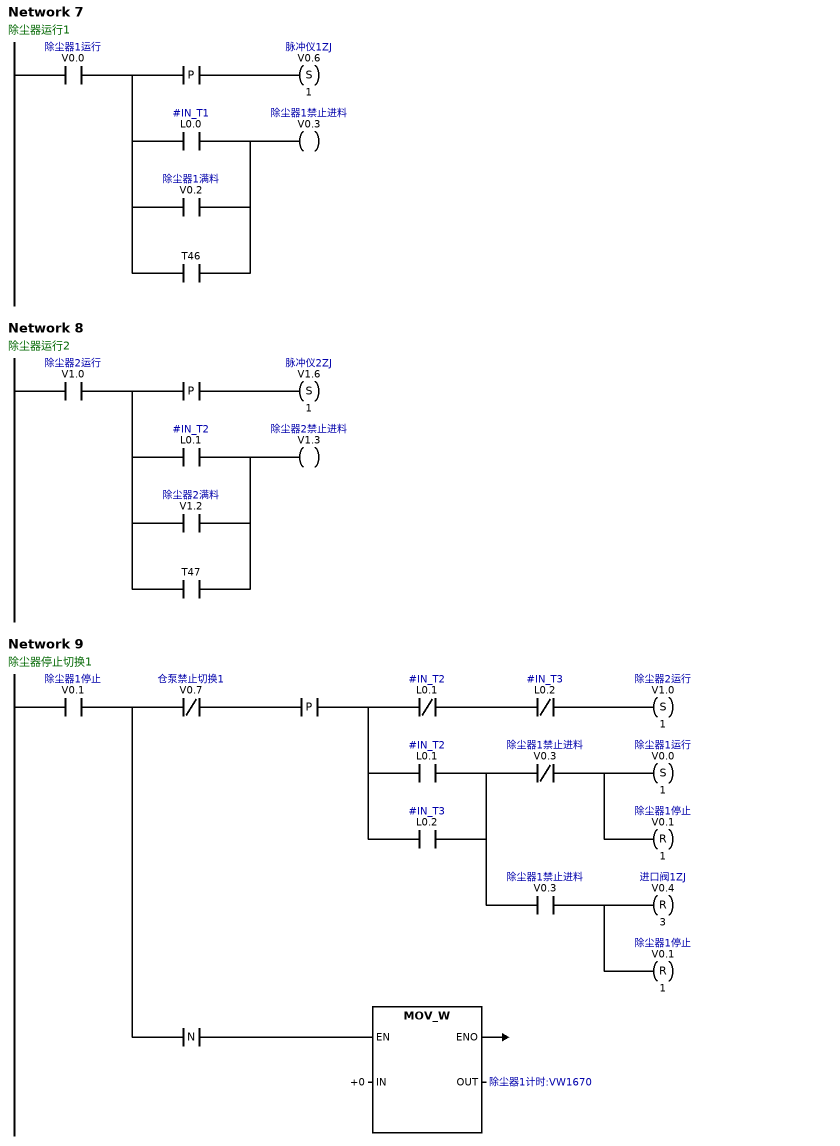
Network 7
// 除尘器运行1
LD     除尘器1运行:V0.0
LPS
EU
S      脉冲仪1ZJ:V0.6, 1
LPP
LD     #IN_T1:L0.0
O      除尘器1满料:V0.2
O      T46
ALD
=      除尘器1禁止进料:V0.3
Network 8
// 除尘器运行2
LD     除尘器2运行:V1.0
LPS
EU
S      脉冲仪2ZJ:V1.6, 1
LPP
LD     #IN_T2:L0.1
O      除尘器2满料:V1.2
O      T47
ALD
=      除尘器2禁止进料:V1.3
Network 9
// 除尘器停止切换1
LD     除尘器1停止:V0.1
LPS
AN     仓泵禁止切换1:V0.7
EU
LPS
AN     #IN_T2:L0.1
AN     #IN_T3:L0.2
S      除尘器2运行:V1.0, 1
LPP
LD     #IN_T2:L0.1
O      #IN_T3:L0.2
ALD
LPS
AN     除尘器1禁止进料:V0.3
S      除尘器1运行:V0.0, 1
R      除尘器1停止:V0.1, 1
LPP
A      除尘器1禁止进料:V0.3
R      进口阀1ZJ:V0.4, 3
R      除尘器1停止:V0.1, 1
LPP
ED
MOVW   +0, 除尘器1计时:VW1670
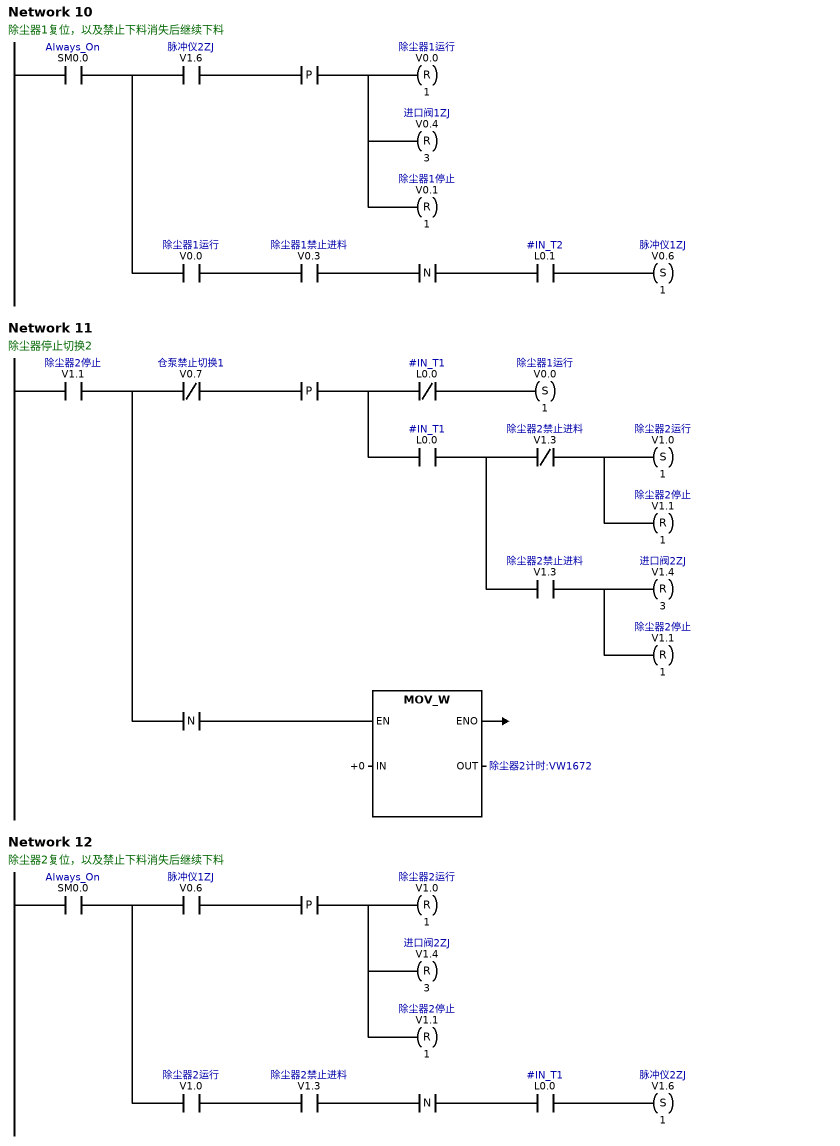
Network 10
// 除尘器1复位，以及禁止下料消失后继续下料
LD     Always_On:SM0.0
LPS
A      脉冲仪2ZJ:V1.6
EU
R      除尘器1运行:V0.0, 1
R      进口阀1ZJ:V0.4, 3
R      除尘器1停止:V0.1, 1
LPP
A      除尘器1运行:V0.0
A      除尘器1禁止进料:V0.3
ED
A      #IN_T2:L0.1
S      脉冲仪1ZJ:V0.6, 1
Network 11
// 除尘器停止切换2
LD     除尘器2停止:V1.1
LPS
AN     仓泵禁止切换1:V0.7
EU
LPS
AN     #IN_T1:L0.0
S      除尘器1运行:V0.0, 1
LPP
A      #IN_T1:L0.0
LPS
AN     除尘器2禁止进料:V1.3
S      除尘器2运行:V1.0, 1
R      除尘器2停止:V1.1, 1
LPP
A      除尘器2禁止进料:V1.3
R      进口阀2ZJ:V1.4, 3
R      除尘器2停止:V1.1, 1
LPP
ED
MOVW   +0, 除尘器2计时:VW1672
Network 12
// 除尘器2复位，以及禁止下料消失后继续下料
LD     Always_On:SM0.0
LPS
A      脉冲仪1ZJ:V0.6
EU
R      除尘器2运行:V1.0, 1
R      进口阀2ZJ:V1.4, 3
R      除尘器2停止:V1.1, 1
LPP
A      除尘器2运行:V1.0
A      除尘器2禁止进料:V1.3
ED
A      #IN_T1:L0.0
S      脉冲仪2ZJ:V1.6, 1
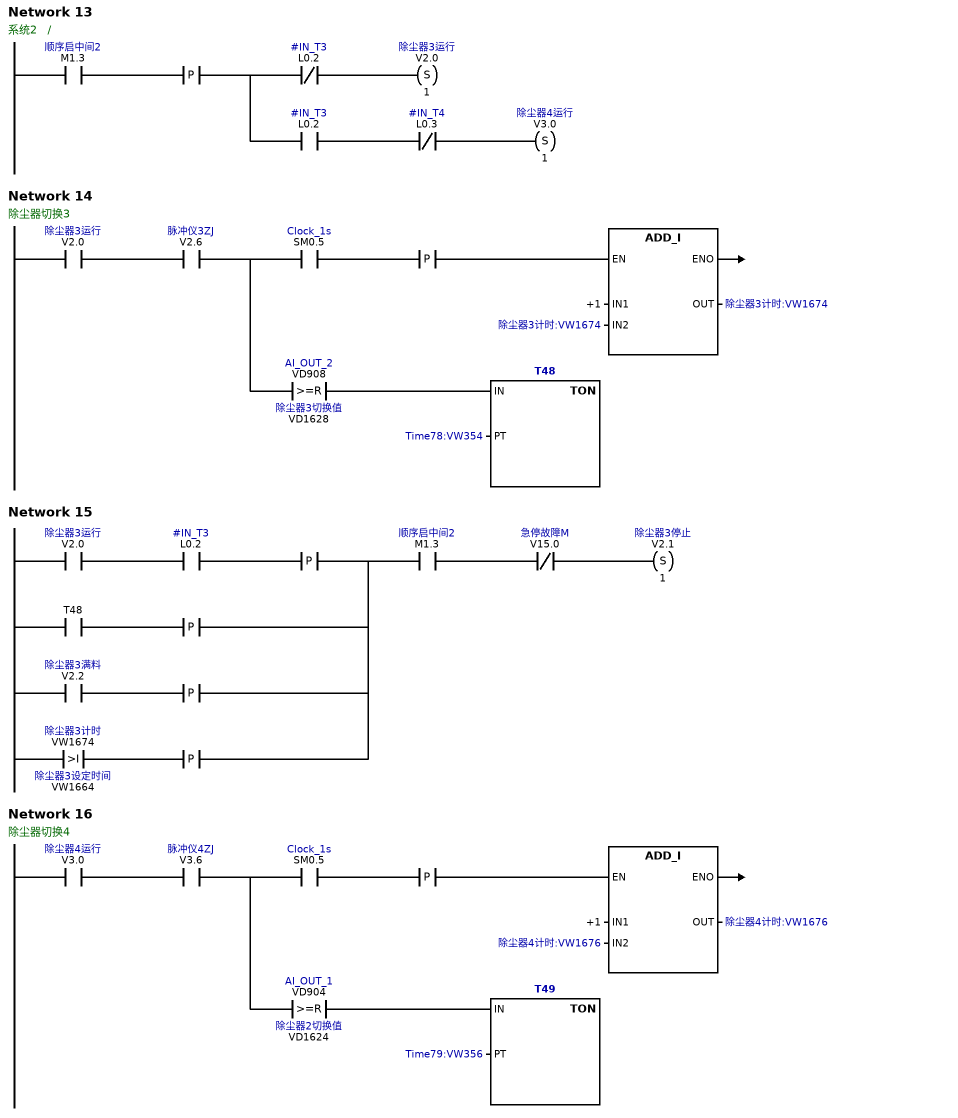
Network 13
// 系统2  
// 
LD     顺序启中间2:M1.3
EU
LPS
AN     #IN_T3:L0.2
S      除尘器3运行:V2.0, 1
LPP
A      #IN_T3:L0.2
AN     #IN_T4:L0.3
S      除尘器4运行:V3.0, 1
Network 14
// 除尘器切换3
LD     除尘器3运行:V2.0
A      脉冲仪3ZJ:V2.6
LPS
A      Clock_1s:SM0.5
EU
+I     +1, 除尘器3计时:VW1674
LPP
AR>=   AI_OUT_2:VD908, 除尘器3切换值:VD1628
TON    T48, Time78:VW354
Network 15
LD     除尘器3运行:V2.0
A      #IN_T3:L0.2
EU
LD     T48
EU
OLD
LD     除尘器3满料:V2.2
EU
OLD
LDW>   除尘器3计时:VW1674, 除尘器3设定时间:VW1664
EU
OLD
A      顺序启中间2:M1.3
AN     急停故障M:V15.0
S      除尘器3停止:V2.1, 1
Network 16
// 除尘器切换4
LD     除尘器4运行:V3.0
A      脉冲仪4ZJ:V3.6
LPS
A      Clock_1s:SM0.5
EU
+I     +1, 除尘器4计时:VW1676
LPP
AR>=   AI_OUT_1:VD904, 除尘器2切换值:VD1624
TON    T49, Time79:VW356
